// Core §7.7(c) — per-root session + enforcement. Login/logout is DATA-DRIVEN
// (§3.10(a')): the HMI writes ReqUser/ReqSecret and pulses ReqLogin/ReqLogout;
// the secret is cleared after every attempt. Policy default: fully open (§7.7(b)).
FUNCTION_BLOCK FB_AccessManager
VAR_INPUT
    ReqUser   : STRING(32);          // HMI-writable login request
    ReqSecret : STRING(32);          // cleared after each attempt (§7.7(c))
    ReqLogin  : BOOL;
    ReqLogout : BOOL;
END_VAR
VAR_OUTPUT
    CurrentUser  : STRING(32);
    CurrentLevel : E_AccessLevel;    // HMI greys controls from this; PLC re-checks
    LoginFailed  : BOOL;             // last attempt outcome (HMI feedback)
END_VAR
VAR PERSISTENT
    Policy : ST_AccessPolicy;        // §3.8a station config; edit gated by ACCESS_POLICY
END_VAR
VAR
    {attribute 'OPC.UA.DA' := '0'}
    _provider : I_AccessProvider;
    {attribute 'OPC.UA.DA' := '0'}
    _log      : POINTER TO FB_AlarmLog;
    _tIdle    : TON;
END_VAR

// event/session handling is in Cyclic (called by the owning Unit each scan)

METHOD Cyclic : BOOL
VAR
    lvl : E_AccessLevel;
    loginHandled : BOOL;
    logoutHandled : BOOL;
END_VAR
loginHandled := ReqLogin;
IF loginHandled THEN
    ReqLogin := FALSE;
    lvl := E_AccessLevel.NONE;
    IF _provider <> 0 THEN
        lvl := _provider.Authenticate(User := ReqUser, Secret := ReqSecret);
    END_IF
    ReqSecret := '';                                   // never retain the secret
    IF lvl > E_AccessLevel.NONE THEN
        CurrentUser := ReqUser;
        CurrentLevel := lvl;
        LoginFailed := FALSE;
        _M_Audit('std.audit.login', CurrentUser);
    ELSE
        LoginFailed := TRUE;
        _M_Audit('std.audit.loginFailed', ReqUser);
    END_IF
END_IF
logoutHandled := ReqLogout;
IF logoutHandled THEN
    ReqLogout := FALSE;
    IF CurrentLevel > E_AccessLevel.NONE THEN
        _M_Audit('std.audit.logout', CurrentUser);
        CurrentUser := '';
        CurrentLevel := E_AccessLevel.NONE;
    END_IF
END_IF
// idle auto-logout (§7.7(c)); any successful login rearms it
_tIdle(IN := (Policy.SessionTimeout > T#0S) AND (CurrentLevel > E_AccessLevel.NONE) AND NOT loginHandled,
       PT := Policy.SessionTimeout);
IF _tIdle.Q THEN
    _M_Audit('std.audit.autoLogout', CurrentUser);
    CurrentUser := '';
    CurrentLevel := E_AccessLevel.NONE;
END_IF
Cyclic := TRUE;
END_METHOD

// Startup/station-configuration seam; runtime HMI writes remain Unit-gated.
METHOD ConfigureRequired : BOOL
VAR_INPUT
    Gate : E_GatedAction;
    Level : E_AccessLevel;
END_VAR
IF (TO_INT(Gate) < 0) OR (TO_INT(Gate) > TO_INT(E_GatedAction.POWER_CONTROL)) THEN
    ConfigureRequired := FALSE;
ELSE
    Policy.Required[TO_INT(Gate)] := Level;
    ConfigureRequired := TRUE;
END_IF
END_METHOD

// ST-facing request seam. OPC UA clients continue to write the published request data.
METHOD RequestLogin : BOOL
VAR_INPUT
    User : STRING(32);
    Secret : STRING(32);
END_VAR
ReqUser := User;
ReqSecret := Secret;
ReqLogin := TRUE;
RequestLogin := TRUE;
END_METHOD

// ST-facing request seam; the cyclic edge handler performs the state change and audit.
METHOD RequestLogout : BOOL
ReqLogout := TRUE;
RequestLogout := TRUE;
END_METHOD

// pure check for UI/logic — no logging
METHOD Permits : BOOL
VAR_INPUT
    Gate : E_GatedAction;
END_VAR
Permits := TO_DINT(CurrentLevel) >= TO_DINT(Policy.Required[TO_INT(Gate)]);
END_METHOD

// gated-entry check: a DENIED attempt is audited as a MESSAGE event (§8.3/§7.7(c))
METHOD PermitsLogged : BOOL
VAR_INPUT
    Gate : E_GatedAction;
END_VAR
PermitsLogged := Permits(Gate := Gate);
IF NOT PermitsLogged THEN
    _M_Audit('std.audit.accessDenied', CurrentUser);
END_IF
END_METHOD

METHOD Setup : BOOL
VAR_INPUT
    Provider : I_AccessProvider;
    pAlarmLog : POINTER TO FB_AlarmLog;
END_VAR
IF Provider <> 0 THEN
    _provider := Provider;                  // Unit OnInit may attach only the audit log
END_IF
_log := pAlarmLog;
Setup := TRUE;
END_METHOD

// audit trail for free: come+gone MESSAGE lands in the §8.3 ring
METHOD PRIVATE _M_Audit
VAR_INPUT
    What : STRING(64);
    Who : STRING(32);
END_VAR
VAR
    auditSlot : INT;
    txt : STRING(255);
END_VAR
IF _log = 0 THEN
    RETURN;
END_IF
txt := CONCAT(What, ': ');
txt := CONCAT(txt, Who);
auditSlot := _log^.Raise(Reason := E_Reason.NONE, Text := txt,
                 Source := 'Access', Severity := E_Severity.LOW,
                 Category := E_Category.SYSTEM, ResetClass := E_ResetClass.AUTO_RESET);
IF auditSlot > 0 THEN
    _log^.Gone(Slot := auditSlot);                     // instant come+gone -> ring entry
END_IF
END_METHOD

END_FUNCTION_BLOCK

(* stored: Version 1.1.0.1, ProductVersion 3.1.4024.12
   POU FB_AccessManager: Id {a5754c56-27d7-4f58-93a7-2bc76040ee69}, SpecialFunc None
   Method Cyclic: Id {f524a87a-e061-4ff8-b535-53d9cf845caa}
   Method ConfigureRequired: Id {ca211e14-0c26-4d31-aaf3-bf00dccfed16}
   Method RequestLogin: Id {126d9072-7c2d-4ed5-978f-501975d1299e}
   Method RequestLogout: Id {2c9e0da4-edd0-461d-a5ce-adcdc0497718}
   Method Permits: Id {0a2e27c0-07c7-4a25-aa9d-77c75345beec}
   Method PermitsLogged: Id {95aa1389-db64-4f1a-8591-0c8cfda5199a}
   Method Setup: Id {380f7b09-d7bf-4407-aa62-ac88c12cd7da}
   Method _M_Audit: Id {4a43a0c7-56fe-4d93-9850-5fda5b3cfdb6} *)
